(* CODESYS project CtaAppInfluxLog_1.0.0.1.library
   Description: Trendlog Library der CTA
   Version: 1.0.0.1
   Title: CtaAppInfluxLog
   Author: SIS
   LanguageModelAttribute: qualified-access-only
   DocFormat: reStructuredText
   Placeholder: CtaAppInfluxLog
   DefaultNamespace: CtaAppInfluxLog
   CompiledLibraryCompatibilityVersion: CODESYS V3.5 SP16 Patch 3
   Company: CTA

Project tree, tasks and I/O mapping:
  libraries: Standard, 3.5.18.0 (System); VisuSymbols, 4.5.0.0 (System); SysFile, 3.5.17.0 (System); SysProcess, 3.5.17.0 (System); StringUtils, 3.5.18.0 (System); Util, 3.5.19.0 (System); CtaSysInfluxLog, 1.0.0.3 (CTA)
  30 Program Organization Units/
    NODE/
      STRING/
        function block FB_LOG_NODE_STRING [ST]: KEY, ENABLE, DESTROYAFTERLOG, SET_VALUE
      BOOL/
        function block FB_LOG_NODE_BOOL [ST]: ENABLE, KEY, DESTROYAFTERLOG, SET_VALUE
      INT/
        function block FB_LOG_NODE_INT [ST]: DESTROYAFTERLOG, SET_VALUE, KEY, ENABLE
      REAL/
        function block FB_LOG_NODE_REAL [ST]: SET_VALUE, DESTROYAFTERLOG, KEY, ENABLE
  00000000-0000-0000-0000-000000000000|D:\CoDeSys\LibrariesV3\trunk\Intern\CAA\CAA Template\3.4.0.0 draft\Placeholder.xml
  00000000-0000-0000-0000-000000000000|D:\CoDeSys\LibrariesV3\trunk\Intern\CAA\CAA Template\3.2.0.3 draft\Prefix.pdf
  00000000-0000-0000-0000-000000000000|D:\CoDeSys\LibrariesV3\trunk\Intern\CAA\CAA Template\3.5.2.0 draft\Placeholder.xml
  20 Structs/
  50 Images/
  10 Documenation/
    global variables VersionHistory
    global variables readMe
  21 Interface/
  11 Library Parameter/
  12 Konstanten/
  13 Globale Variablen/
  text list GlobalTextList
  22 Enumeration/
*)

// 10 Documenation/VersionHistory
(* 

.. image:: ../../Images/CTA_Logo.jpg
   :align: right
   :width: 15% 

**Vorlage**   


============ =========== =========== ============================================
**Date**     **Version** **Author**  **Change**
------------ ----------- ----------- --------------------------------------------
04.03.2021   0.0.0.0     SIS         Vorlage erstellt

============ =========== =========== ============================================


*)
VAR_GLOBAL
    stInfo : STRING:= '0.0.0.0, Vorlage, CTA';
END_VAR

// 10 Documenation/readMe
(*

**ReadMe**

|	**Empfehlung**
|
|	Für das Trendloggen in die InfluxDb wird nachfolgender Code benötigt.                           
|	Zusätzlich muss im PLC_PRG der Fb fbLibAp94_1InfluxDb als Funktionsbaustein Instanziert werden.
|  
|
| *Beispiel* 

 ============= ================================================================================================================================
 Beschreibung  Code                                                                                                
 ============= ================================================================================================================================                   
 Pou oder SmFb .. code-block:: codesys
 
                    // Deklaration der Struktur Variable scInfluxData
                    VAR
                        scInfluxData                    :   WagoAppInfluxDB.typInfluxField;
                    END_VAR     

                    (* Code als actInfluxDb *)
                    // Clear Data
                        scInfluxData.sKey   := '';
                        scInfluxData.sValue := '';
                    // Write Data
                        scInfluxData.sKey   := CONCAT(STR1 := stObjID, STR2 := '_xOn');
                        scInfluxData.sValue := TO_STRING(xOn); 
                        scInfluxData.eType  := WagoAppInfluxDB.eFieldValueType.eFVT_BOOL;
                        LibAp94InfluxDb.gvlLibAp94_1InfluxDb.fbLibAp94_2DataCollecter.proInfluxDbData := scInfluxData;
                    // Clear Data
                        scInfluxData.sKey   := '';
                        scInfluxData.sValue := '';
                    // Write Data
                        scInfluxData.sKey   := CONCAT(STR1 := stObjID, STR2 := '_rOnY');
                        scInfluxData.sValue := TO_STRING(rOnY); 
                        scInfluxData.eType  := WagoAppInfluxDB.eFieldValueType.eFVT_FLOAT;
                        LibAp94InfluxDb.gvlLibAp94_1InfluxDb.fbLibAp94_2DataCollecter.proInfluxDbData := scInfluxData;    
                    // Clear Data
                        scInfluxData.sKey   := '';
                        scInfluxData.sValue := '';
                    // Write Data
                        scInfluxData.sKey   := CONCAT(STR1 := stObjID, STR2 := '_xError');
                        scInfluxData.sValue := TO_STRING(proLockDown); 
                        scInfluxData.eType  := WagoAppInfluxDB.eFieldValueType.eFVT_BOOL;
                        LibAp94InfluxDb.gvlLibAp94_1InfluxDb.fbLibAp94_2DataCollecter.proInfluxDbData := scInfluxData;           
                                                                                                                                                                 
 ============= ================================================================================================================================ 
*)
VAR_GLOBAL
    xReadMeDone              :   BOOL;
END_VAR

// 30 Program Organization Units/NODE/STRING/FB_LOG_NODE_STRING
FUNCTION_BLOCK FB_LOG_NODE_STRING 
VAR
	ITF_LOG_NODE_STRING	:	CtaSysInfluxLog.ITF_LOG_NODE_STRING;
	xNoMem				:	BOOL;
END_VAR

PROPERTY KEY : STRING(255)
GET
IF __QUERYINTERFACE(ITF_LOG_NODE_STRING,ITF_LOG_NODE_STRING) THEN
	KEY := ITF_LOG_NODE_STRING.KEY;
END_IF;
END_GET
SET
IF __QUERYINTERFACE(ITF_LOG_NODE_STRING,ITF_LOG_NODE_STRING) THEN
	ITF_LOG_NODE_STRING.KEY := KEY;
END_IF;
END_SET
END_PROPERTY

PROPERTY ENABLE : BOOL
SET
VAR
	xSema	:	BOOL;
END_VAR
IF ENABLE AND ITF_LOG_NODE_STRING = 0 AND NOT xNoMem AND CtaSysInfluxLog.GVL_TREND.FB_INFLUX_NODE_FACTORY.READY THEN
	ITF_LOG_NODE_STRING := CtaSysInfluxLog.GVL_TREND.FB_INFLUX_NODE_FACTORY.GET_STRING_LOG_NODE(xSema => xSema);
	IF NOT xSema THEN
		IF __QUERYINTERFACE(ITF_LOG_NODE_STRING,ITF_LOG_NODE_STRING) THEN
			ITF_LOG_NODE_STRING.ENABLE := TRUE;
		ELSE
			xNoMem					:= TRUE;		
		END_IF;
	ELSE
		RETURN;
	END_IF;
ELSIF NOT ENABLE THEN
	IF __QUERYINTERFACE(ITF_LOG_NODE_STRING,ITF_LOG_NODE_STRING) THEN
		ITF_LOG_NODE_STRING.ENABLE 	:= FALSE;
		ITF_LOG_NODE_STRING 		:= 0;
		xNoMem						:= FALSE;	
	END_IF;
END_IF;
END_SET
GET
IF __QUERYINTERFACE(ITF_LOG_NODE_STRING,ITF_LOG_NODE_STRING) THEN
	ENABLE := ITF_LOG_NODE_STRING.ENABLE;
ELSE
	ENABLE := FALSE;
END_IF;
END_GET
END_PROPERTY

PROPERTY DESTROYAFTERLOG : BOOL
SET
IF __QUERYINTERFACE(ITF_LOG_NODE_STRING,ITF_LOG_NODE_STRING) THEN
	ITF_LOG_NODE_STRING.DESTROYAFTERLOG := DESTROYAFTERLOG;
	ITF_LOG_NODE_STRING := 0;
END_IF;
END_SET
END_PROPERTY

PROPERTY SET_VALUE : STRING(250)
SET
IF __QUERYINTERFACE(ITF_LOG_NODE_STRING,ITF_LOG_NODE_STRING) THEN
	ITF_LOG_NODE_STRING.SET_VALUE := SET_VALUE;
END_IF;
END_SET
END_PROPERTY

END_FUNCTION_BLOCK

// 30 Program Organization Units/NODE/BOOL/FB_LOG_NODE_BOOL
FUNCTION_BLOCK FB_LOG_NODE_BOOL
VAR
	ITF_LOG_NODE_BOOL	:	CtaSysInfluxLog.ITF_LOG_NODE_BOOL;
	xNoMem				:	BOOL;
END_VAR

PROPERTY ENABLE : BOOL
SET
VAR
	xSema	:	BOOL;
END_VAR
IF ENABLE AND ITF_LOG_NODE_BOOL = 0 AND NOT xNoMem AND CtaSysInfluxLog.GVL_TREND.FB_INFLUX_NODE_FACTORY.READY THEN
	ITF_LOG_NODE_BOOL := CtaSysInfluxLog.GVL_TREND.FB_INFLUX_NODE_FACTORY.GET_BOOL_LOG_NODE(xSema => xSema);
	IF NOT xSema THEN
		IF __QUERYINTERFACE(ITF_LOG_NODE_BOOL,ITF_LOG_NODE_BOOL) THEN
			ITF_LOG_NODE_BOOL.ENABLE := TRUE;
		ELSE
			xNoMem					:= TRUE;	
		END_IF;
	ELSE
		RETURN;
	END_IF;
ELSIF NOT ENABLE THEN
	IF __QUERYINTERFACE(ITF_LOG_NODE_BOOL,ITF_LOG_NODE_BOOL) THEN
		ITF_LOG_NODE_BOOL.ENABLE := FALSE;
		ITF_LOG_NODE_BOOL		 := 0;
		xNoMem					 := FALSE;
	END_IF;
END_IF;
END_SET
GET
IF __QUERYINTERFACE(ITF_LOG_NODE_BOOL,ITF_LOG_NODE_BOOL) THEN
	ENABLE := ITF_LOG_NODE_BOOL.ENABLE;
ELSE
	ENABLE := FALSE;
END_IF;
END_GET
END_PROPERTY

PROPERTY KEY : STRING(255)
GET
IF __QUERYINTERFACE(ITF_LOG_NODE_BOOL,ITF_LOG_NODE_BOOL) THEN
	KEY := ITF_LOG_NODE_BOOL.KEY;
END_IF;
END_GET
SET
IF __QUERYINTERFACE(ITF_LOG_NODE_BOOL,ITF_LOG_NODE_BOOL) THEN
	ITF_LOG_NODE_BOOL.KEY := KEY;
END_IF;
END_SET
END_PROPERTY

PROPERTY DESTROYAFTERLOG : BOOL
SET
IF __QUERYINTERFACE(ITF_LOG_NODE_BOOL,ITF_LOG_NODE_BOOL) THEN
	ITF_LOG_NODE_BOOL.DESTROYAFTERLOG := DESTROYAFTERLOG;
	ITF_LOG_NODE_BOOL := 0;
END_IF;
END_SET
END_PROPERTY

PROPERTY SET_VALUE : BOOL
SET
IF __QUERYINTERFACE(ITF_LOG_NODE_BOOL,ITF_LOG_NODE_BOOL) THEN
	ITF_LOG_NODE_BOOL.SET_VALUE := SET_VALUE;
END_IF;
END_SET
END_PROPERTY

END_FUNCTION_BLOCK

// 30 Program Organization Units/NODE/INT/FB_LOG_NODE_INT
FUNCTION_BLOCK FB_LOG_NODE_INT
VAR
	ITF_LOG_NODE_INT	:	CtaSysInfluxLog.ITF_LOG_NODE_INT;
	xNoMem				:	BOOL;
END_VAR

PROPERTY DESTROYAFTERLOG : BOOL
SET
IF __QUERYINTERFACE(ITF_LOG_NODE_INT,ITF_LOG_NODE_INT) THEN
	ITF_LOG_NODE_INT.DESTROYAFTERLOG := DESTROYAFTERLOG;
	ITF_LOG_NODE_INT := 0;
END_IF;
END_SET
END_PROPERTY

PROPERTY SET_VALUE : INT
SET
IF __QUERYINTERFACE(ITF_LOG_NODE_INT,ITF_LOG_NODE_INT) THEN
	ITF_LOG_NODE_INT.SET_VALUE := SET_VALUE;
END_IF;
END_SET
END_PROPERTY

PROPERTY KEY : STRING(255)
GET
IF __QUERYINTERFACE(ITF_LOG_NODE_INT,ITF_LOG_NODE_INT) THEN
	KEY := ITF_LOG_NODE_INT.KEY;
END_IF;
END_GET
SET
IF __QUERYINTERFACE(ITF_LOG_NODE_INT,ITF_LOG_NODE_INT) THEN
	ITF_LOG_NODE_INT.KEY := KEY;
END_IF;
END_SET
END_PROPERTY

PROPERTY ENABLE : BOOL
SET
VAR
	xSema	:	BOOL;
END_VAR
IF ENABLE AND ITF_LOG_NODE_INT = 0 AND NOT xNoMem AND CtaSysInfluxLog.GVL_TREND.FB_INFLUX_NODE_FACTORY.READY THEN
	ITF_LOG_NODE_INT := CtaSysInfluxLog.GVL_TREND.FB_INFLUX_NODE_FACTORY.GET_INT_LOG_NODE(xSema => xSema);
	IF NOT xSema THEN
		IF __QUERYINTERFACE(ITF_LOG_NODE_INT,ITF_LOG_NODE_INT) THEN
			ITF_LOG_NODE_INT.ENABLE := TRUE;
		ELSE
			xNoMem					:= TRUE;
		END_IF;
	ELSE
		RETURN;
	END_IF;
ELSIF NOT ENABLE THEN
	IF __QUERYINTERFACE(ITF_LOG_NODE_INT,ITF_LOG_NODE_INT) THEN
		ITF_LOG_NODE_INT.ENABLE := FALSE;
		ITF_LOG_NODE_INT 		:= 0;
		xNoMem					:= FALSE;
	END_IF;
END_IF;
END_SET
GET
IF __QUERYINTERFACE(ITF_LOG_NODE_INT,ITF_LOG_NODE_INT) THEN
	ENABLE := ITF_LOG_NODE_INT.ENABLE;
ELSE
	ENABLE := FALSE;
END_IF;
END_GET
END_PROPERTY

END_FUNCTION_BLOCK

// 30 Program Organization Units/NODE/REAL/FB_LOG_NODE_REAL
FUNCTION_BLOCK FB_LOG_NODE_REAL
VAR
	ITF_LOG_NODE_REAL	:	CtaSysInfluxLog.ITF_LOG_NODE_REAL;
	xNoMem				:	BOOL;
END_VAR

PROPERTY SET_VALUE : REAL
SET
IF __QUERYINTERFACE(ITF_LOG_NODE_REAL,ITF_LOG_NODE_REAL) THEN
	ITF_LOG_NODE_REAL.SET_VALUE := SET_VALUE;
END_IF;
END_SET
END_PROPERTY

PROPERTY DESTROYAFTERLOG : BOOL
SET
IF __QUERYINTERFACE(ITF_LOG_NODE_REAL,ITF_LOG_NODE_REAL) THEN
	ITF_LOG_NODE_REAL.DESTROYAFTERLOG := DESTROYAFTERLOG;
	ITF_LOG_NODE_REAL := 0;
END_IF;
END_SET
END_PROPERTY

PROPERTY KEY : STRING(255)
GET
IF __QUERYINTERFACE(ITF_LOG_NODE_REAL,ITF_LOG_NODE_REAL) THEN
	KEY := ITF_LOG_NODE_REAL.KEY;
END_IF;
END_GET
SET
IF __QUERYINTERFACE(ITF_LOG_NODE_REAL,ITF_LOG_NODE_REAL) THEN
	ITF_LOG_NODE_REAL.KEY := KEY;
END_IF;
END_SET
END_PROPERTY

PROPERTY ENABLE : BOOL
SET
VAR
	xSema	:	BOOL;
END_VAR
IF ENABLE AND ITF_LOG_NODE_REAL = 0 AND NOT xNoMem AND CtaSysInfluxLog.GVL_TREND.FB_INFLUX_NODE_FACTORY.READY THEN
	ITF_LOG_NODE_REAL := CtaSysInfluxLog.GVL_TREND.FB_INFLUX_NODE_FACTORY.GET_REAL_LOG_NODE(xSema => xSema);
	IF NOT xSema THEN
		IF __QUERYINTERFACE(ITF_LOG_NODE_REAL,ITF_LOG_NODE_REAL) THEN
			ITF_LOG_NODE_REAL.ENABLE := TRUE;
		ELSE
			xNoMem					:= TRUE;		
		END_IF;
	ELSE
		RETURN;
	END_IF;
ELSIF NOT ENABLE THEN
	IF __QUERYINTERFACE(ITF_LOG_NODE_REAL,ITF_LOG_NODE_REAL) THEN
		ITF_LOG_NODE_REAL.ENABLE := FALSE;
		ITF_LOG_NODE_REAL 		 := 0;
		xNoMem					 := FALSE;
	END_IF;
END_IF;
END_SET
GET
IF __QUERYINTERFACE(ITF_LOG_NODE_REAL,ITF_LOG_NODE_REAL) THEN
	ENABLE := ITF_LOG_NODE_REAL.ENABLE;
ELSE
	ENABLE := FALSE;
END_IF;
END_GET
END_PROPERTY

END_FUNCTION_BLOCK
